FUNCTION_BLOCK ABS_VALUE
VAR_INPUT
    InputVal : INT;    // Input integer value
END_VAR

VAR_OUTPUT
    Result : INT;      // Output integer: absolute value of InputVal (always 0 or positive)
END_VAR

VAR CONSTANT
    MAX_INT  : INT := 16#7FFF;     // Maximum INT value (32767)
    MIN_SAFE : INT := -16#7FFF;     // -32767; any value less than this must be the extreme negative
END_VAR

// Compute absolute value with saturation for the problematic input
IF InputVal < MIN_SAFE THEN
    Result := MAX_INT;           // For the extreme value (i.e. only -32768 is less than -32767)
ELSIF InputVal < 0 THEN
    Result := -InputVal;         // For a normal negative value, negate it
ELSE
    Result := InputVal;          // For zero or positive values, no change is needed
END_IF;

END_FUNCTION_BLOCK